FUNCTION_BLOCK FB_PackMLModule EXTENDS FB_PackMLModeSet
VAR_INPUT
END_VAR
VAR_OUTPUT
END_VAR
VAR
END_VAR

END_FUNCTION_BLOCK

(* stored: Version 1.1.0.1, ProductVersion 3.1.4026.18
   POU FB_PackMLModule: Id {e5d0f60c-8d1a-48c8-9daa-cfbe39692472}, SpecialFunc None *)
